FUNCTION_BLOCK FB_FallibleINT IMPLEMENTS I_FallibleINT
VAR
    bError : BOOL;
    sErrorMsg : T_MaxString;
    nVal : INT;
END_VAR

METHOD ClearError

bError := FALSE;
sErrorMsg := '';
END_METHOD

METHOD GetError : BOOL

GetError := bError;
END_METHOD

METHOD GetErrorMsg : Tc2_System.T_MaxString

GetErrorMsg := sErrorMsg;
END_METHOD


METHOD SetError
VAR_INPUT
    sMsg	: Tc2_System.T_MaxString;
END_VAR

bError := TRUE;
sErrorMsg := sMsg;
END_METHOD

PROPERTY Val : INT
GET

Val := nVal;
END_GET
SET

nVal := Val;
END_SET
END_PROPERTY

END_FUNCTION_BLOCK

(* stored: Version 1.1.0.1, ProductVersion 3.1.4022.18
   POU FB_FallibleINT: Id {1f018dee-e093-42d6-aac2-80dec4064397}, SpecialFunc None
   Method ClearError: Id {dde3723b-7aaa-417e-81c5-b16ac78d4e3f}
   Method GetError: Id {3e5299e2-fa75-465f-b800-efb06043c86d}
   Method GetErrorMsg: Id {e19e5c01-ba06-40c7-9626-250e60887447}
   Method SetError: Id {4849cc0b-5ccb-453c-85a1-d142ca83e883}
   Property Val: Id {e8414c8b-d29c-418d-be0b-54bb442f2ab8}
   Get Get: Id {d3588344-3245-4a23-925d-a695ac01e428}
   Set Set: Id {ea00948a-beec-47a2-bcce-561de83e256d} *)
